FUNCTION_BLOCK TcMessage_Ext IMPLEMENTS ITcMessage_Ext
VAR_INPUT
END_VAR
VAR_OUTPUT
END_VAR
VAR
    fbMsg : FB_TcMessage; 
	fbTest : Tc3_EventLogger.FB_TcEvent;
	fbInfo : Tc3_EventLogger.FB_TcSourceInfo;
	_loggerLevel : TcEventSeverity := TcEventSeverity.Info;
END_VAR

PROPERTY PUBLIC LoggerLevel : TcEventSeverity
GET
LoggerLevel := _loggerLevel;
END_GET
SET
_loggerLevel := LoggerLevel;
END_SET
END_PROPERTY

METHOD PUBLIC Send : BOOL
VAR_INPUT
	eventType : Tc3_EventLogger.TcEventEntry;
	args : STRING(255);
END_VAR
IF eventType.eSeverity >= LoggerLevel THEN
	THIS^.fbMsg.CreateEx(eventType, 0);
	THIS^.fbMsg.ipArguments.AddString(args);
	THIS^.fbMsg.Send(0);
	THIS^.fbMsg.Release();
END_IF
END_METHOD

END_FUNCTION_BLOCK

(* stored: Version 1.1.0.1, ProductVersion 3.1.4024.11
   POU TcMessage_Ext: Id {fba85ae3-7e59-4012-8e9f-d6b698999416}, SpecialFunc None
   Property LoggerLevel: Id {d4dda1b0-5cf3-4c00-a006-c2d92bc1d845}
   Get Get: Id {cb24dbdf-44c6-4307-94b5-8bb6b5c77333}
   Set Set: Id {7f7479d9-f690-4591-be8b-69e28cbe99d5}
   Method Send: Id {59b43c0a-c63f-4ea7-9f49-bd3f6e5004ae} *)
